// TwinCAT 3 PLC project Untitled1
// ProgramVersion: 3.1.4022.7
// libraries:
//   LCLS Vacuum, * (SLAC - LCLS)
//   LCLSVacuumSerialDriverLib, * (SLAC - LCLS)
//   Tc2_SerialCom, * (Beckhoff Automation GmbH)
//   Tc2_Standard, * (Beckhoff Automation GmbH)
//   Tc2_System, * (Beckhoff Automation GmbH)
//   Tc3_Module, * (Beckhoff Automation GmbH)
// project tree:
//   GVLs/ GVL_COM.TcGVL (not stored), GVL_Devices.TcGVL
//   / PlcTask.TcTTO
//   POUs/ MAIN.TcPOU, PRG_COM.TcPOU
// real-time tasks:
//   TASK PlcTask: cycle T#10ms, priority 20, ADS port 350

CONFIGURATION Untitled1
    RESOURCE PLC ON TwinCAT3
        TASK PlcTask(INTERVAL := T#10ms, PRIORITY := 20);
        PROGRAM MAIN WITH PlcTask : MAIN;
    END_RESOURCE
END_CONFIGURATION

// ---- GVLs/GVL_Devices.TcGVL
VAR_GLOBAL
	
	// non serial interface
	{attribute 'TcLinkTo':=  '.i_xAtSpd := TIIB[Box 2 (EP2338-0002)]^Channel 1^Input;
							.i_xFaultNC := TIIB[Box 2 (EP2338-0002)]^Channel 2^Input;
							.q_PumpingStation := TIIB[Box 7 (EP2624-0002)]^Channel 1^Output'}

	PTM : FB_PTM_Pfeiffer;
	
	(*Pfeiffer*)
	// They share the same serial port
	st_Pfeiffer_CTRL 			: ARRAY[1..20] OF ST_PfeifferControl;
	st_Pfeiffer_RBK 			: ARRAY[1..20] OF ST_PfeifferStatus;
	fb_PfeifferCom : FB_PFEIFFER_COM;
	
END_VAR

// ---- POUs/MAIN.TcPOU
PROGRAM MAIN
VAR
{attribute 'TcLinkTo' := 'TIIB[Box 7 (EP2624-0002)]^Channel 1^Output'}	
x_PumpStation AT %Q*	:	BOOL;
{attribute 'TcLinkTo' := 'TIIB[Box 7 (EP2624-0002)]^Channel 2^Output'}
x_ErrorReset AT %Q*	:	BOOL;
{attribute 'TcLinkTo' := 'TIIB[Box 2 (EP2338-0002)]^Channel 1^Input'}
x_AtSpeed AT %I*	:	BOOL;
{attribute 'TcLinkTo' := 'TIIB[Box 2 (EP2338-0002)]^Channel 2^Input'}
x_FaultNC AT %I*	:	BOOL;

END_VAR

//Pfeiffer Turbo
(* Instanitate the Function block for Pump Control*)
PTM(i_xExtIlkOK:= TRUE , iq_stPTM=> );

(*Assign adresses to the pfeiffer controllers connected to this serial terminal*)
st_Pfeiffer_CTRL[1].iSerialAddress :=1;
st_Pfeiffer_CTRL[1].xEnableComm := TRUE;
	
(* Instanitate the Function block for serial communication with Pfeiffer*)	
fb_PfeifferCom(astPfeifferControl := st_Pfeiffer_CTRL,
			   astPfeifferStatus:= st_Pfeiffer_RBK,
				SerialRXBuffer:= E2_SerialRXBuffer,
				SerialTXBuffer:= E2_SerialTXBuffer);
				

(* Copy Status Pv's into the PTM structure*)
PTM.M_Serial_IO(st_Pfeiffer_CTRL[1],st_Pfeiffer_RBK[1]);

END_PROGRAM

// ---- POUs/PRG_COM.TcPOU
PROGRAM PRG_COM
VAR
END_VAR

//needs to run on a seperate task
//PTM_01
(*Instanitate Serial port com function *) 
fbSerialLineControl(
	Mode:= SERIALLINEMODE_EL6_22B,
	pComIn:= ADR(stComIn),
	pComOut:=ADR(stComOut),
	SizeComIn:= SIZEOF(stComIn),
	TxBuffer:= SerialRXBuffer,
	RxBuffer:= SerialTXBuffer,
	Error=> ,
	ErrorID=> );
	
(*
//PTM_02 and PTM_03
(*Instanitate Serial port com function *) 
E2_fbSerialLineControl(
	Mode:= SERIALLINEMODE_EL6_22B,
	pComIn:= ADR(E2_stComIn),
	pComOut:=ADR(E2_stComOut),
	SizeComIn:= SIZEOF(E2_stComIn),
	TxBuffer:= E2_SerialRXBuffer,
	RxBuffer:= E2_SerialRXBuffer,
	Error=> ,
	ErrorID=> );*)

END_PROGRAM
